    previousSetPos : LREAL; // degrees
    previousSetVelo : LREAL; // degrees/sec
    previousSetAcc : LREAL; // degrees/sec2

    deltaTime : LREAL; // seconds
    
    nextSetPosMax : LREAL;
    nextSetPosMin : LREAL;
    
    nextSetVeloMax : LREAL;
    nextSetVeloMin : LREAL;
    
    nextSetAccMax : LREAL;
    nextSetAccMin : LREAL;
    
    
    lastReceivedDcTime : LINT;
    cycle : INT;
    secondsAfterNewUpdate : LREAL;
    MAX_NUMBER_OF_CYCLES : INT;
    
    minPositionSetpoint : LREAL;
    maxPositionSetpoint : LREAL;
    
END_VAR


// calculate which cycle we are after receiving new updates from the slalib task
IF cycle > MAX_NUMBER_OF_CYCLES THEN 
    cycle := 0; // should not be happening, don't extrapolate
ELSIF  dcTime > lastReceivedDcTime THEN
    // OK we received new values from the slalib task!
    lastReceivedDcTime := dcTime;
    cycle := 0;
ELSE
    cycle := cycle + 1;
END_IF 

secondsAfterNewUpdate := cycle * TIME_TO_LREAL(GLOBAL.config.PLC_FAST_TASK_TIME) / 1000.0;  // TIME_TO_LREAL returns milliseconds!


IF _requestSynchronize THEN    
    physical.PlcToNc.ExtSetPos := physical.NcToPlc.ActPos;
    physical.PlcToNc.ExtSetVelo := 0.0;
    physical.PlcToNc.ExtSetAcc := 0.0;
    
    previousSetPos := physical.PlcToNc.ExtSetPos;
    previousSetVelo := physical.PlcToNc.ExtSetVelo;
    previousSetAcc := physical.PlcToNc.ExtSetAcc;
    
    _requestSynchronize := FALSE;
ELSIF _requestSetPosition THEN
    physical.PlcToNc.ExtSetPos := _requestSetPositionValue;
    physical.PlcToNc.ExtSetVelo := 0.0;
    physical.PlcToNc.ExtSetAcc := 0.0;
    
    previousSetPos := _requestSetPositionValue;
    previousSetVelo := 0.0;
    previousSetAcc := 0.0;
    
    _requestSetPosition := FALSE;      

ELSIF _requestStartTracking THEN
    tracking := TRUE;
    _requestStartTracking := FALSE;
ELSIF _requestStopTracking THEN
    tracking := FALSE;
    _requestStopTracking := FALSE;
ELSE
    
    
    // we expect MAX_VELOCITY and MAX_ACCELERATION to be positive values!
    velocityLimit := ABS(velocityLimit);
    accelerationLimit := ABS(accelerationLimit);
    
    previousSetPos := physical.PlcToNc.ExtSetPos;
    previousSetVelo := physical.PlcToNc.ExtSetVelo;
    previousSetAcc := physical.PlcToNc.ExtSetAcc;
    
    IF tracking THEN
        
        physical.PlcToNc.ExtSetPos  := virtual.NcToPlc.SetPos  + targetPos - trackingStart;
        physical.PlcToNc.ExtSetVelo := virtual.NcToPlc.SetVelo + targetVelo; 
        physical.PlcToNc.ExtSetAcc  := virtual.NcToPlc.SetAcc  + targetAcc;
        
        // The PLC FAST task runs faster than the C++ Slalib task.
        // As a result, the targetPos/targetVelo/targetAcc are updated at a slower rate than the axis setpoints,
        // which means that the axes setpoints versus time look like a "stair" instead of a smooth curve.
        // Therefore, we extrapolate the position setpoint, based on the velocity of the axes
        // The residual position errors are neglegible 
        
        IF cycle > 0 THEN
            // p(t) = p0 + v*t + (a*t^2)/2
            physical.PlcToNc.ExtSetPos := physical.PlcToNc.ExtSetPos 
                                          + targetVelo * secondsAfterNewUpdate
                                          + targetAcc * secondsAfterNewUpdate*secondsAfterNewUpdate / 2.0; 
        END_IF
        
        minPositionSetpoint := minTrackingPositionSetpoint;
        maxPositionSetpoint := maxTrackingPositionSetpoint;
        
    ELSE
        
        physical.PlcToNc.ExtSetPos  := virtual.NcToPlc.SetPos;
        physical.PlcToNc.ExtSetVelo := virtual.NcToPlc.SetVelo; 
        physical.PlcToNc.ExtSetAcc  := virtual.NcToPlc.SetAcc;
        
        minPositionSetpoint := minVirtualPositionSetpoint;
        maxPositionSetpoint := maxVirtualPositionSetpoint;
    END_IF
    
    
    // check if the position limit is reached
    //=======================================================================================
    // we can still go a bit over it, because otherwise the axis would stop very abruptly.
    limitReached := (physical.PlcToNc.ExtSetPos < minPositionSetpoint) OR (physical.PlcToNc.ExtSetPos > maxPositionSetpoint);
    IF limitReached THEN
        physical.PlcToNc.ExtSetPos := LIMIT(minPositionSetpoint, physical.PlcToNc.ExtSetPos, maxPositionSetpoint);
	END_IF
    
    
    
    // Limit the setpoint trajectory!!!!
    //=======================================================================================
    
    deltaTime := TIME_TO_LREAL(GLOBAL.config.PLC_FAST_TASK_TIME) / 1000.0;
    
    // calculate the min/max acceleration for the next setpoint
    nextSetAccMax := accelerationLimit;  // we don't take jerk into account
    nextSetAccMin := -accelerationLimit; // we don't take jerk into account:
    
    // calculate the min/max velocity for the next setpoint
    nextSetVeloMax := LIMIT(-velocityLimit, previousSetVelo + nextSetAccMax * deltaTime, velocityLimit);
    nextSetVeloMin := LIMIT(-velocityLimit, previousSetVelo + nextSetAccMin * deltaTime, velocityLimit);
    
    // calculate the next min/max position
    nextSetPosMax := previousSetPos + nextSetVeloMax * deltaTime;
    nextSetPosMin := previousSetPos + nextSetVeloMin * deltaTime;
    
    // now update the setpoint generator values
    physical.PlcToNc.ExtSetPos  := LIMIT(nextSetPosMin  , physical.PlcToNc.ExtSetPos  , nextSetPosMax);
    physical.PlcToNc.ExtSetVelo := LIMIT(nextSetVeloMin , physical.PlcToNc.ExtSetVelo , nextSetVeloMax);
    physical.PlcToNc.ExtSetAcc  := LIMIT(nextSetAccMin  , physical.PlcToNc.ExtSetAcc  , nextSetAccMax);
    
    // Set the direction
    //===================
    IF physical.PlcToNc.ExtSetPos > physical.NcToPlc.ActPos THEN
        physical.PlcToNc.ExtSetDirection := 1;
    ELSIF physical.PlcToNc.ExtSetPos < physical.NcToPlc.ActPos THEN
        physical.PlcToNc.ExtSetDirection := -1;
    ELSE
        physical.PlcToNc.ExtSetDirection := 0;
    END_IF
    (*
    IF physical.PlcToNc.ExtSetVelo > 0 THEN
        physical.PlcToNc.ExtSetDirection := 1;
    ELSIF physical.PlcToNc.ExtSetVelo < 0 THEN
        physical.PlcToNc.ExtSetDirection := -1;
    ELSE
        physical.PlcToNc.ExtSetDirection := 0;
    END_IF
    *)

END_IF

METHOD stopTracking : BOOL
VAR_INPUT
END_VAR
_requestStopTracking := TRUE;
END_METHOD

METHOD FB_init : BOOL
VAR_INPUT
	bInitRetains : BOOL; // if TRUE, the retain variables are initialized (warm start / cold start)
	bInCopyCode : BOOL;  // if TRUE, the instance afterwards gets moved into the copy code (online change)
END_VAR
IF TIME_TO_LREAL(GLOBAL.config.PLC_FAST_TASK_TIME) > 0 THEN  // watch for division by zero
    MAX_NUMBER_OF_CYCLES := LREAL_TO_INT( TIME_TO_LREAL(GLOBAL.config.SLALIB_TASK_TIME) / TIME_TO_LREAL(GLOBAL.config.PLC_FAST_TASK_TIME) );
END_IF
END_METHOD

METHOD startTracking : BOOL
VAR_INPUT
END_VAR
_requestStartTracking := TRUE;
END_METHOD

METHOD setPosition
VAR_INPUT
    value : LREAL;
END_VAR
_requestSetPosition := TRUE;
_requestSetPositionValue := value;
END_METHOD

METHOD synchronize
VAR_INPUT
END_VAR
_requestSynchronize := TRUE;
END_METHOD

END_FUNCTION_BLOCK

// ---- MTCS/Common/StateMachines/AngularAxis.TcPOU
FUNCTION_BLOCK AngularAxis EXTENDS SM_AngularAxis;
VAR_INPUT
END_VAR
VAR_OUTPUT
END_VAR
VAR
    _testVar : BOOL;
END_VAR

SUPER^();

END_FUNCTION_BLOCK

// ---- MTCS/Axes/Helper/AxesUnlockBrakeHelper.TcPOU
FUNCTION_BLOCK AxesUnlockBrakeHelper
VAR_INPUT
END_VAR
VAR_OUTPUT
END_VAR
VAR_IN_OUT
    unlockBrake : AxesUnlockBrakeProcess;
    driveChannel : AX52XXDriveChannel;
END_VAR
VAR
    _ton : TON;
    _seconds : LREAL;
    _formatString : FB_FormatString;
    _msg : STRING;
END_VAR

IF unlockBrake.isBusy() THEN
    
    IF NOT unlockBrake.isStarted() THEN
        unlockBrake._state := 0;
        unlockBrake.setStarted();
	END_IF
    
    CASE unlockBrake._state OF
        0:
            unlockBrake.setActualStatus('Unlocking brake'); 
            driveChannel.processes.setBrake.start(DriveBrakeStates.BRAKE_FORCE_UNLOCK);
            unlockBrake._state := 1;
        1:
            IF driveChannel.processes.setBrake.isIdle() THEN
                IF driveChannel.processes.setBrake.isGood() THEN
                    _ton(IN := FALSE);
                    _ton(IN := TRUE, PT := LREAL_TO_TIME(unlockBrake.get.seconds * 1000.0));
                    unlockBrake._state := 2;
                ELSE
                    unlockBrake._state := 999;
                    unlockBrake.setActualStatus('Could not change brake to FORCE UNLOCK'); 
				END_IF
			END_IF
        2:
            _ton(IN := TRUE);
            IF _ton.Q THEN
                unlockBrake._state := 3;
            ELSE
                _seconds := TIME_TO_LREAL(_ton.ET) / 1000.0;
                _formatString(sFormat := 'Waiting for %.1fs...', arg1 := F_LREAL(_seconds), sOut => _msg);
                unlockBrake.setActualStatus(_msg); 
			END_IF
        3:
            unlockBrake.setActualStatus('Setting brake to auto'); 
            driveChannel.processes.setBrake.start(DriveBrakeStates.BRAKE_AUTOMATIC);
            unlockBrake._state := 4;
        4:
            IF driveChannel.processes.setBrake.isIdle() THEN
                IF driveChannel.processes.setBrake.isGood() THEN
                    unlockBrake.setActualStatus('Done, brake set to AUTO again'); 
                    unlockBrake._state := 1000;
                ELSE
                    unlockBrake.setActualStatus('Could not change brake to AUTO!!! Brake is still UNLOCKED!!!'); 
                    unlockBrake._state := 999;
				END_IF
			END_IF

        999:
            unlockBrake.setBad();
            unlockBrake.setFinished();
        1000:
            unlockBrake.setGood();
            unlockBrake.setFinished();
        
    END_CASE
    
END_IF

END_FUNCTION_BLOCK

// ---- MTCS/Common/StateMachines/AX52XXDriveChannel.TcPOU
FUNCTION_BLOCK AX52XXDriveChannel EXTENDS SM_AX52XXDriveChannel
VAR_INPUT
END_VAR
VAR_OUTPUT
END_VAR
VAR
    _pointerToAxisRef : POINTER TO AXIS_REF := 0;
    _SoERead : FB_SoERead;
    _SoEWrite : FB_SoEWrite;
    _SoEReset : FB_SoEReset;
	_safetyErrorAckTon: TON;
END_VAR

_update();

isInSafetate := safetyOptionState.0;

_updating();
_reading();
_writing();
_resetting();
_settingBrake();
_acknowledgeSafetyError();

_update();

METHOD _resetting
VAR_INPUT
END_VAR

IF processes.reset.isBusy() THEN
    
    IF NOT processes.reset.isStarted() THEN
        processes.reset._state := 0;
        processes.reset.setStarted();
	END_IF
    
    CASE processes.reset._state OF
        0:  
            processes.reset.setActualStatus('Resetting any errors');
            // Execute must be FALSE first, to make sure we can create a rising edge
            _SoEReset(
                NetId := '',
                Execute := FALSE,
                Axis := _pointerToAxisRef^);
            _SoEReset(
                NetId := '',
                Execute := TRUE,
                Axis := _pointerToAxisRef^,
                Timeout := T#10S); // From Beckhoff help pages: "The timeout time must be 10s, because the reset can take up to 10s."
            processes.reset._state := 1;
        1:
            _SoEReset(
                NetId := '',
                Execute := TRUE,
                Axis := _pointerToAxisRef^,
                Timeout := T#10S);
            
            IF _SoEReset.Error THEN
                processes.reset.setActualStatus(
                        CONCAT(    
                               CONCAT('Reset error: AdsErrId=', UINT_TO_STRING(_SoEReset.AdsErrId)), 
                               CONCAT(' SercosErrId=', UINT_TO_STRING(_SoEReset.SercosErrId))
                        )
                );
                processes.reset.adsErrorId := _SoEReset.AdsErrId;
                processes.reset.sercosErrorId := _SoEReset.SercosErrId;
                processes.reset._state := 999;
            ELSIF NOT _SoEReset.Busy THEN
                // ok done!
                processes.reset._state := 1000;
            END_IF
        999:
            // error!
            processes.reset.setBad();
            processes.reset.setFinished();
        1000:
            // all done!
            processes.reset.setActualStatus('Reset finished');
            processes.reset.setGood();
            processes.reset.setFinished();
    
	END_CASE
        

END_IF
END_METHOD

METHOD _reading
VAR_INPUT
END_VAR
VAR
    valueAddress : PVOID;
END_VAR
IF processes.read.statuses.busyStatus.busy THEN
    
    IF processes.read.get.noOfBytes = 1 THEN
        valueAddress := ADR(processes.read.value1Byte);
        processes.read.setGood();
    ELSIF processes.read.get.noOfBytes = 2 THEN
        valueAddress := ADR(processes.read.value2Bytes);
        processes.read.setGood();
    ELSIF processes.read.get.noOfBytes = 4 THEN
        valueAddress := ADR(processes.read.value4Bytes);
        processes.read.setGood();
    ELSE
        processes.read.setBad();
        processes.read.setFinished();
	END_IF
    
    IF _pointerToAxisRef = 0 THEN
        processes.read.setActualStatus('Internal bug: axis_ref not set');
        processes.read.setBad();
        processes.read.setFinished();
	END_IF
    
    IF processes.read.statuses.healthStatus.good THEN
         
        IF NOT processes.read.statuses.startedStatus.started THEN
            // make sure we get a rising edge
            _SoERead(Execute := FALSE, Axis:= _pointerToAxisRef^);
            
            (* execute the SoE read command *)
            _SoERead(
                NetId    := '',
                Idn      :=  processes.read.get.index,
                Element  := EC_SOE_ELEMENT_VALUE,
                pDstBuf  := valueAddress,
                BufLen   := processes.read.get.noOfBytes,
                Execute  := TRUE,
                Timeout  := DEFAULT_ADS_TIMEOUT,
                Axis     := _pointerToAxisRef^);
            
             processes.read.setStarted();
             
		END_IF
        
       (* Make sure the Execute input is reset *)
        _SoERead(Execute := FALSE, Axis:= _pointerToAxisRef^);
        
        (* update the health status *)
        SUPER^.processes.read.statuses.healthStatus(isGood := NOT _SoERead.Error);
        
        (* update the busy status *)
        SUPER^.processes.read.statuses.busyStatus(isBusy := _SoERead.Busy);
        
        (* update the error ID *)
        SUPER^.processes.read.adsErrorId := _SoERead.AdsErrId;
        SUPER^.processes.read.sercosErrorId := _SoERead.SercosErrId;
             
	END_IF
 
END_IF
END_METHOD

METHOD _acknowledgeSafetyError
VAR_INPUT
END_VAR

VAR
END_VAR

IF processes.acknowledgeSafetyError.isBusy() THEN
    
    IF NOT processes.acknowledgeSafetyError.isStarted() THEN
        processes.acknowledgeSafetyError._state := 0;
        processes.acknowledgeSafetyError.setStarted();
	END_IF
    
    CASE processes.acknowledgeSafetyError._state OF
        0:  
            processes.acknowledgeSafetyError.setActualStatus('Commanding safety card');
            safetyErrorAck := TRUE;
            _safetyErrorAckTon(IN := FALSE);
            
            processes.acknowledgeSafetyError._state := 1;
        1:
            _safetyErrorAckTon(IN := TRUE, PT := T#0.3S);
            IF _safetyErrorAckTon.Q THEN
                processes.acknowledgeSafetyError._state := 2;
            END_IF
        2:
            safetyErrorAck := FALSE;
            _safetyErrorAckTon(IN := FALSE);
            processes.acknowledgeSafetyError._state := 3;
        3:
            _safetyErrorAckTon(IN := TRUE, PT := T#0.3S);
            IF _safetyErrorAckTon.Q THEN
                processes.acknowledgeSafetyError._state := 4;
            END_IF
        4:
            safetyErrorAck := TRUE;
            _safetyErrorAckTon(IN := FALSE);
            processes.acknowledgeSafetyError._state := 5;
        5:
            _safetyErrorAckTon(IN := TRUE, PT := T#0.3S);
            IF _safetyErrorAckTon.Q THEN
                processes.acknowledgeSafetyError._state := 6;
            END_IF
        6:
            safetyErrorAck := FALSE;
            _safetyErrorAckTon(IN := FALSE);
            _safetyErrorAckTon(IN := TRUE, PT := T#1S);
            processes.acknowledgeSafetyError._state := 7;
        7:
            _safetyErrorAckTon(IN := TRUE, PT := T#1S);
            IF _safetyErrorAckTon.Q THEN
                IF isInSafetate THEN
                    processes.acknowledgeSafetyError._state := 999;
                    processes.acknowledgeSafetyError.setActualStatus('Safe state persists!');
                ELSE
                    processes.acknowledgeSafetyError._state := 1000;
                    processes.acknowledgeSafetyError.setActualStatus('Drive unblocked by safety');
                END_IF
            
			END_IF
        999:
            // error!
            processes.acknowledgeSafetyError.setBad();
            processes.acknowledgeSafetyError.setFinished();
        1000:
            // all done!
            processes.acknowledgeSafetyError.setGood();
            processes.acknowledgeSafetyError.setFinished();
    
        END_CASE
            

END_IF
END_METHOD

METHOD _updating
VAR_INPUT
END_VAR

IF processes.update.isBusy() THEN
    
    IF NOT processes.update.isStarted() THEN
        processes.update._state := 0;
        processes.update.setStarted();
	END_IF
    
    CASE processes.update._state OF
        0:  
            processes.update.setActualStatus('Reading P-0-0092 Configured channel peak current');
            processes.read.start(index := P_0_IDN + 92, noOfBytes := 4);
            processes.update._state := 1;
        1:
            IF processes.read.isIdle() THEN
                IF processes.read.isGood() THEN
                    channelPeakCurrent(newAmpsValue := UDINT_TO_LREAL(processes.read.value4Bytes) / 1000.0);
                    processes.update._state := 2;
                ELSE
                    processes.update.setActualStatus('Could not read P-0-0092');
                    processes.update._state := 999;
				END_IF
            END_IF
        2:
            processes.update.setActualStatus('Reading P-0-0093 Configured channel current');
            processes.read.start(index := P_0_IDN + 93, noOfBytes := 4);
            processes.update._state := 3;
        3:
            IF processes.read.isIdle() THEN
                IF processes.read.isGood() THEN
                    channelRatedCurrent(newAmpsValue := UDINT_TO_LREAL(processes.read.value4Bytes) / 1000.0);
                    processes.update._state := 4;
                ELSE
                    processes.update.setActualStatus('Could not read P-0-0093');
                    processes.update._state := 999;
				END_IF
            END_IF
        4:  
            processes.update.setActualStatus('Reading P-0-0070 Motor continuous stall torque');
            processes.read.start(index := P_0_IDN + 70, noOfBytes := 2);
            processes.update._state := 5;
        5:
            IF processes.read.isIdle() THEN
                IF processes.read.isGood() THEN
                        continuousStallTorque(newNewtonmeterValue := UINT_TO_LREAL(processes.read.value2Bytes) / 100.0);
                        processes.update._state := 6;
                ELSE
                    processes.update.setActualStatus('Could not read P-0-070');
                    processes.update._state := 999;
				END_IF
            END_IF 
        6:  
            processes.update.setActualStatus('Reading S-0-0111 Motor continuous stall current');
            processes.read.start(index := S_0_IDN + 111, noOfBytes := 4);
            processes.update._state := 7;
        7:
            IF processes.read.isIdle() THEN
                IF processes.read.isGood() THEN
                        continuousStallCurrent(newAmpsValue := UDINT_TO_LREAL(processes.read.value4Bytes) / 1000.0);
                        processes.update._state := 8;
                ELSE
                    processes.update.setActualStatus('Could not read S-0-0111');
                    processes.update._state := 999;
				END_IF
            END_IF
        8:
            // now we can simply calculate the torque constant:
            // but watch for division by zero!!!
            IF continuousStallCurrent.amps.value > 0 THEN
                torqueConstant := continuousStallTorque.newtonmeter.value / continuousStallCurrent.amps.value;
                processes.update._state := 9;
            ELSE
                torqueConstant := 0.0;
                processes.update.setActualStatus('Torque constant cannot be calculated!');
                processes.update._state := 999;
			END_IF
        9:
            processes.update.setActualStatus('Reading S-0-0082 Positive torque limit value');
            processes.read.start(index := S_0_IDN + 82, noOfBytes := 2);
            processes.update._state := 10;
        10:
            IF processes.read.isIdle() THEN
                IF processes.read.isGood() THEN
                        positiveTorqueLimit(
                            newFractionValue := UINT_TO_LREAL(processes.read.value2Bytes) / 1000.0, 
                            maxNewtonmeter   := channelPeakCurrent.amps.value * torqueConstant);
                        processes.update._state := 11;
                ELSE
                    processes.update.setActualStatus('Could not read S-0-0082');
                    processes.update._state := 999;
				END_IF
            END_IF 
        11:  
            processes.update.setActualStatus('Reading S-0-0083 Negative torque limit value');
            processes.read.start(index := S_0_IDN + 83, noOfBytes := 2);
            processes.update._state := 12;
        12:
            IF processes.read.isIdle() THEN
                IF processes.read.isGood() THEN
                        negativeTorqueLimit(
                            newFractionValue := UINT_TO_LREAL(processes.read.value2Bytes) / 1000.0, 
                            maxNewtonmeter   := channelPeakCurrent.amps.value * torqueConstant);
                        processes.update._state := 13;
                ELSE
                    processes.update.setActualStatus('Could not read S-0-0082');
                    processes.update._state := 999;
				END_IF
            END_IF
        13:  
            processes.update.setActualStatus('Reading S-0-0092 Bipolar torque limit value');
            processes.read.start(index := S_0_IDN + 92, noOfBytes := 2);
            processes.update._state := 14;
        14:
            IF processes.read.isIdle() THEN
                IF processes.read.isGood() THEN
                        bipolarTorqueLimit(
                            newFractionValue := UINT_TO_LREAL(processes.read.value2Bytes) / 1000.0, 
                            maxNewtonmeter   := channelPeakCurrent.amps.value * torqueConstant);
                        processes.update._state := 15;
                ELSE
                    processes.update.setActualStatus('Could not read S-0-0092');
                    processes.update._state := 999;
				END_IF
            END_IF       
        15:  
            processes.update.setActualStatus('Reading P-0-0096 Motor control word');
            processes.read.start(index := P_0_IDN + 96, noOfBytes := 2);
            processes.update._state := 16;
        16:
            IF processes.read.isIdle() THEN
                IF processes.read.isGood() THEN
                    IF processes.read.value2Bytes.0 THEN
                       brakeState := DriveBrakeStates.BRAKE_FORCE_LOCK;
                    ELSIF processes.read.value2Bytes.1 THEN
                       brakeState := DriveBrakeStates.BRAKE_FORCE_UNLOCK;
                    ELSE
                       brakeState := DriveBrakeStates.BRAKE_AUTOMATIC;
                    END_IF
                    brakeStateDescription := DriveBrakeStatesToString(brakeState);
                    processes.update._state := 17;
                ELSE
                    processes.update.setActualStatus('Could not read P-0-0096');
                    processes.update._state := 999;
				END_IF
            END_IF     
        17:  
            processes.update.setActualStatus('Reading S-0-0032 Primary operation mode');
            processes.read.start(index := S_0_IDN + 32, noOfBytes := 2);
            processes.update._state := 18;
        18:
            IF processes.read.isIdle() THEN
                IF processes.read.isGood() THEN
                    IF processes.read.value2Bytes = 0 THEN
                       operatingMode := DriveOperatingModes.OPERATING_MODE_NONE;
                    ELSIF    processes.read.value2Bytes = 1
                          OR processes.read.value2Bytes = 32769 THEN
                       operatingMode := DriveOperatingModes.OPERATING_MODE_TORQUE_CONTROL;
                    ELSIF    processes.read.value2Bytes = 2
                          OR processes.read.value2Bytes = 32770 THEN
                       operatingMode := DriveOperatingModes.OPERATING_MODE_VELOCITY_CONTROL;
                    ELSIF    processes.read.value2Bytes = 3
                          OR processes.read.value2Bytes = 4
                          OR processes.read.value2Bytes = 11
                          OR processes.read.value2Bytes = 12
                          OR processes.read.value2Bytes = 32771
                          OR processes.read.value2Bytes = 32772
                          OR processes.read.value2Bytes = 32779
                          OR processes.read.value2Bytes = 32780 THEN
                       operatingMode := DriveOperatingModes.OPERATING_MODE_POSITION_CONTROL;
                    ELSE
                       operatingMode := DriveOperatingModes.OPERATING_MODE_NONE;
                    END_IF
                    operatingModeDescription := DriveOperatingModesToString(operatingMode);
                    processes.update._state := 19;
                ELSE
                    processes.update.setActualStatus('Could not read S-0-0032');
                    processes.update._state := 999;
				END_IF
            END_IF
        19:
            // all done
            processes.update._state := 1000;
        999:
            // error!
            processes.update.setBad();
            processes.update.setFinished();
        1000:
            // all done!
            processes.update.setActualStatus('Updated');
            processes.update.setGood();
            processes.update.setFinished();
    
    
	END_CASE
        

END_IF
END_METHOD

METHOD _settingBrake
VAR_INPUT
END_VAR
VAR
    ctrlWord : WORD := 0;
END_VAR

IF processes.setBrake.isBusy() THEN
    
    IF NOT processes.setBrake.isStarted() THEN
        processes.setBrake._state := 0;
        processes.setBrake.setStarted();
	END_IF
    
    CASE processes.setBrake._state OF
        0:  
            processes.setBrake.setActualStatus(CONCAT('Setting brake ', DriveBrakeStatesToString(processes.setBrake.get.newState)));          
            CASE processes.setBrake.get.newState OF
               DriveBrakeStates.BRAKE_FORCE_LOCK:
                    ctrlWord.0 := TRUE;
                    ctrlWord.1 := FALSE;
               DriveBrakeStates.BRAKE_FORCE_UNLOCK:
                    ctrlWord.0 := FALSE;
                    ctrlWord.1 := TRUE;
               DriveBrakeStates.BRAKE_AUTOMATIC:
                    ctrlWord.0 := FALSE;
                    ctrlWord.1 := FALSE;
            END_CASE
            
            processes.write.start(index := P_0_IDN + 96, noOfBytes := 2, value1Byte := 0, value2Bytes := ctrlWord, value4Bytes := 0);
            processes.setBrake._state := 1;
        1:
            IF processes.write.isIdle() THEN
                IF processes.write.isGood() THEN
                    processes.setBrake._state := 2;
                ELSE
                    processes.setBrake.setActualStatus('Could not write P-0-0096');
                    processes.setBrake._state := 999;
				END_IF
            END_IF    
        2:  
            processes.setBrake.setActualStatus('Reading P-0-0096 Motor control word');
            processes.read.start(index := P_0_IDN + 96, noOfBytes := 2);
            processes.setBrake._state := 3;
        3:
            IF processes.read.isIdle() THEN
                IF processes.read.isGood() THEN
                    IF processes.read.value2Bytes.0 THEN
                       brakeState := DriveBrakeStates.BRAKE_FORCE_LOCK;
                    ELSIF processes.read.value2Bytes.1 THEN
                       brakeState := DriveBrakeStates.BRAKE_FORCE_UNLOCK;
                    ELSE
                       brakeState := DriveBrakeStates.BRAKE_AUTOMATIC;
                    END_IF
                    brakeStateDescription := DriveBrakeStatesToString(brakeState);
                    processes.setBrake._state := 1000;
                ELSE
                    processes.setBrake.setActualStatus('Could not read P-0-0096');
                    processes.setBrake._state := 999;
				END_IF
            END_IF     
            

        999:
            // error!
            processes.setBrake.setBad();
            processes.setBrake.setFinished();
        1000:
            // all done!
            processes.setBrake.setActualStatus(CONCAT('Brake now ', brakeStateDescription));
            processes.setBrake.setGood();
            processes.setBrake.setFinished();
    
	END_CASE
        

END_IF
END_METHOD

METHOD _update
VAR_INPUT
END_VAR
SUPER^();

IF statuses.healthStatus.good THEN
    IF statuses.busyStatus.idle THEN
        IF isInSafetate THEN
            actualStatus := 'In safe state';
        ELSE
            actualStatus := 'Idle';
        END_IF
    ELSIF statuses.busyStatus.busy THEN
        actualStatus := 'Busy';
    ELSE
        actualStatus := 'Good';
    END_IF
ELSIF statuses.healthStatus.warning THEN
    IF isInSafetate THEN
        actualStatus := 'SAFE STATE';
    ELSE
        actualStatus := 'Warning';
	END_IF
ELSIF statuses.healthStatus.bad THEN
    IF errorC1D <> 0 THEN
        actualStatus := CONCAT(CONCAT('C1D error (id: ', INT_TO_STRING(errorC1D)), ')');
    ELSIF isInSafetate THEN
        actualStatus := 'SAFE STATE';
    ELSE
        actualStatus := 'ERROR';
	END_IF
ELSE
    actualStatus := '';
END_IF
END_METHOD

METHOD setInternalAxisRef
VAR_INPUT
    pointerToAxisRef : POINTER TO AXIS_REF;
END_VAR
_pointerToAxisRef := pointerToAxisRef;
END_METHOD

METHOD _writing
VAR_INPUT
END_VAR
VAR
    srcAddress : PVOID;
END_VAR
IF processes.write.statuses.busyStatus.busy THEN
    
    IF processes.write.get.noOfBytes = 1 THEN
        srcAddress := ADR(processes.write.get.value1Byte);
        processes.write.setGood();
    ELSIF processes.write.get.noOfBytes = 2 THEN
        srcAddress := ADR(processes.write.get.value2Bytes);
        processes.write.setGood();
    ELSIF processes.write.get.noOfBytes = 4 THEN
        srcAddress := ADR(processes.write.get.value4Bytes);
        processes.write.setGood();
    ELSE
        processes.write.setBad();
        processes.write.setFinished();
	END_IF
     
    IF _pointerToAxisRef = 0 THEN
        processes.write.setActualStatus('Internal bug: axis_ref not set');
        processes.write.setBad();
        processes.write.setFinished();
	END_IF
    
    IF processes.write.statuses.healthStatus.good THEN
         
        IF NOT processes.write.statuses.startedStatus.started THEN
        
            // make sure we get a rising edge
            _SoEWrite(Execute := FALSE, Axis:= _pointerToAxisRef^);
            (* execute the SoE write command *)
            _SoEWrite(
                NetId    := '',
                Idn      :=  processes.write.get.index,
                Element  := EC_SOE_ELEMENT_VALUE,
                pSrcBuf  := srcAddress,
                BufLen   := processes.write.get.noOfBytes,
                Execute  := TRUE,
                Timeout  := DEFAULT_ADS_TIMEOUT,
                Axis     := _pointerToAxisRef^);
            
             processes.write.setStarted();
        ELSE
            // make sure the Exectute input is reset
            _SoEWrite(Execute := FALSE, Axis:= _pointerToAxisRef^);
        
        (* update the health status *)
        SUPER^.processes.write.statuses.healthStatus(isGood := NOT _SoEWrite.Error);
        
        (* update the busy status *)
        SUPER^.processes.write.statuses.busyStatus(isBusy := _SoEWrite.Busy);
        
        (* update the error ID *)
        SUPER^.processes.write.adsErrorId := _SoEWrite.AdsErrId;
        SUPER^.processes.write.sercosErrorId := _SoEWrite.SercosErrId;
		END_IF
        
             
	END_IF
    

 
END_IF
END_METHOD

END_FUNCTION_BLOCK

// ---- MTCS/Common/StateMachines/Current.TcPOU
FUNCTION_BLOCK Current EXTENDS SM_Current
VAR_INPUT
END_VAR
VAR_OUTPUT
END_VAR
VAR
    _testVar : INT;
END_VAR

SUPER^();

END_FUNCTION_BLOCK

// ---- MTCS/Common/HelperCode/DriveBrakeStatesToString.TcPOU
FUNCTION DriveBrakeStatesToString : STRING
VAR_INPUT
    state : DriveBrakeStates;
END_VAR
VAR
END_VAR

CASE state OF
    
    DriveBrakeStates.BRAKE_AUTOMATIC:
        DriveBrakeStatesToString := 'Automatic';
    DriveBrakeStates.BRAKE_FORCE_LOCK:
        DriveBrakeStatesToString := 'Forced LOCK';
    DriveBrakeStates.BRAKE_FORCE_UNLOCK:
        DriveBrakeStatesToString := 'Forced UNLOCK';

END_CASE

END_FUNCTION

// ---- MTCS/Common/HelperCode/DriveOperatingModesToString.TcPOU
FUNCTION DriveOperatingModesToString : STRING
VAR_INPUT
    mode : DriveOperatingModes;
END_VAR
VAR
END_VAR

CASE mode OF
    
    DriveOperatingModes.OPERATING_MODE_NONE:
        DriveOperatingModesToString := 'None';
    DriveOperatingModes.OPERATING_MODE_TORQUE_CONTROL:
        DriveOperatingModesToString := 'Torque control';
    DriveOperatingModes.OPERATING_MODE_VELOCITY_CONTROL:
        DriveOperatingModesToString := 'Velocity control';
    DriveOperatingModes.OPERATING_MODE_POSITION_CONTROL:
        DriveOperatingModesToString := 'Position control';

END_CASE

END_FUNCTION

// ---- MTCS/Common/StateMachines/Force.TcPOU
FUNCTION_BLOCK Force EXTENDS SM_Force
VAR_INPUT
END_VAR
VAR_OUTPUT
END_VAR
VAR
    _testVar : INT;
END_VAR

SUPER^();

END_FUNCTION_BLOCK

// ---- MTCS/Axes/Helper/HMS_TO_DEG.TcPOU
FUNCTION HMS_TO_DEG : LREAL
VAR_INPUT
    positive : BOOL;
    hours : LREAL;
    minutes : LREAL;
    seconds : LREAL;
END_VAR
VAR
END_VAR

HMS_TO_DEG := (hours/24.0 + minutes/(24.0*60.0) + seconds/(24.0*60.0*60.0)) * 360.0;

IF NOT positive THEN
    HMS_TO_DEG := -HMS_TO_DEG;
END_IF

END_FUNCTION

// ---- MTCS/Axes/Helper/DMS_TO_DEG.TcPOU
FUNCTION DMS_TO_DEG : LREAL
VAR_INPUT
    positive : BOOL;
    degrees : LREAL;
    minutes : LREAL;
    seconds : LREAL;
END_VAR
VAR
END_VAR

DMS_TO_DEG := degrees + minutes/60.0 + seconds/3600.0;

IF NOT positive THEN
    DMS_TO_DEG := -DMS_TO_DEG;
END_IF

END_FUNCTION

// ---- MTCS/Axes/Helper/AverageAndRmsCalculator.TcPOU
FUNCTION_BLOCK AverageAndRmsCalculator
VAR_INPUT
    in : LREAL;
END_VAR
VAR_OUTPUT
    avg : LREAL;
    rms : LREAL;
END_VAR
VAR
	_executeMovingAverage : BOOL;
    _ctrl_moving_avg : FB_CTRL_MOVING_AVERAGE;
    _PARAMS : ST_CTRL_MOVING_AVERAGE_PARAMS;
    _array : ARRAY [1..100] OF LREAL;
    
    i : INT := 0;
    sumOfSquares : LREAL := 0.0;
END_VAR


_params.nSamplesToFilter  := 100;
_params.tCtrlCycleTime    := GLOBAL.config.PLC_CTRL_TIME;
_params.tTaskCycleTime    := GLOBAL.config.PLC_TASK_TIME;
_params.pWorkArray_ADR    := ADR(_array);
_params.nWorkArray_SIZEOF := SIZEOF(_array);

IF _executeMovingAverage <> GLOBAL.config.PLC_TASK_FLIP THEN
	_executeMovingAverage := GLOBAL.config.PLC_TASK_FLIP;
	_ctrl_moving_avg(
		fIn             := in,
		fManSyncValue   := 0.0,
		bSync           := FALSE,
		eMode           := E_CTRL_MODE.eCTRL_MODE_ACTIVE,
		bHold           := FALSE,
		stParams        := _params);
    
    sumOfSquares := 0.0;
    FOR i := 1 TO 100 BY 1 DO
        sumOfSquares := sumOfSquares + _array[i]*_array[i];
    END_FOR 
    
    avg := _ctrl_moving_avg.fOut;
    rms := SQRT(sumOfSquares / 100.0);
END_IF

END_FUNCTION_BLOCK

// ---- MTCS/Axes/Helper/AxesCalculateLidaAveragePosition.TcPOU
FUNCTION AxesCalculateLidaAveragePosition : LREAL
VAR_INPUT
    lida1Position : LREAL;
    lida2Position : LREAL;
    lida3Position : LREAL;
    lida4Position : LREAL;
    useLida1 : BOOL;
    useLida2 : BOOL;
    useLida3 : BOOL;
    useLida4 : BOOL;
END_VAR
VAR_OUTPUT
    error : BOOL;
END_VAR
VAR
    sumOfPositions : LREAL := 0.0;
    noOfLidasUsed : INT := 0;
END_VAR

IF useLida1 THEN
    noOfLidasUsed := noOfLidasUsed + 1;
    sumOfPositions := sumOfPositions + lida1Position;
END_IF

IF useLida2 THEN
    noOfLidasUsed := noOfLidasUsed + 1;
    sumOfPositions := sumOfPositions + lida2Position;
END_IF

IF useLida3 THEN
    noOfLidasUsed := noOfLidasUsed + 1;
    sumOfPositions := sumOfPositions + lida3Position;
END_IF

IF useLida4 THEN
    noOfLidasUsed := noOfLidasUsed + 1;
    sumOfPositions := sumOfPositions + lida4Position;
END_IF

// watch for division by zero!
error := noOfLidasUsed = 0;

IF error THEN
    AxesCalculateLidaAveragePosition := 0.0;
ELSE
    AxesCalculateLidaAveragePosition := sumOfPositions / noOfLidasUsed;
END_IF

END_FUNCTION

// ---- MTCS/Axes/Helper/AxesLidaValueToPosition.TcPOU
FUNCTION AxesLidaValueToPosition : LREAL
VAR_INPUT
    id : AxesIds;
    encoderValue : UDINT; 
    invert : BOOL;
END_VAR
VAR
    BITS_PER_TELESCOPE_REVOLUTION : LREAL;
    ENCODER_DIRECTION_INVERSE : BOOL;
END_VAR



IF GLOBAL.config.SIMULATION_ACTIVE THEN
    
    CASE id OF
        AxesIds.AZI:
            BITS_PER_TELESCOPE_REVOLUTION := 3000    // bits per simulation encoder revolution
                                             * 4     // quadrature interpolation
                                             * 1440; // reduction
        AxesIds.ELE:
            BITS_PER_TELESCOPE_REVOLUTION := 3000    // bits per simulation encoder revolution
                                             * 4     // quadrature interpolation
                                             * 1440; // reduction
	END_CASE
ELSE
    
    CASE id OF
        AxesIds.AZI:
            BITS_PER_TELESCOPE_REVOLUTION := 45000    // marks (lines, ticks) on the linear Heidenhain encoder
                                             * 100    // Heidenhain EXE interpolation
                                             * 4;     // quadrature interpolation
        AxesIds.ELE:
            BITS_PER_TELESCOPE_REVOLUTION := 45000    // marks (lines, ticks) on the linear Heidenhain encoder
                                             * 100    // Heidenhain EXE interpolation
                                             * 4;     // quadrature interpolation
	END_CASE

END_IF

    
// we go from unsigned raw value, to signed position in degrees:
IF encoderValue.31 THEN
    AxesLidaValueToPosition := (UDINT_TO_LREAL(encoderValue) - 4294967296) / BITS_PER_TELESCOPE_REVOLUTION * 360.0;  // (rawValue bits - 2**32 bits) / BITS_PER_TELESCOPE_REVOLUTION * 360.0 degrees
ELSE
    AxesLidaValueToPosition := UDINT_TO_LREAL(encoderValue) / BITS_PER_TELESCOPE_REVOLUTION * 360.0; // rawValue bits / BITS_PER_TELESCOPE_REVOLUTION * 360.0 degrees
END_IF

IF invert THEN
    AxesLidaValueToPosition := -AxesLidaValueToPosition;
END_IF

END_FUNCTION

// ---- MTCS/Axes/Helper/AxesSSIValueToPosition.TcPOU
FUNCTION AxesSSIValueToPosition : LREAL
VAR_INPUT
    reduction : LREAL;
    encoderValue : UDINT;
    zeroOffset : LREAL;
END_VAR
VAR
    BITS_PER_ENCODER_REVOLUTION : LREAL := 8192; // 13-bit
    ENCODER_BIT_RANGE : LREAL := 33554432; // 25-bit
END_VAR

// we go from unsigned raw value, to signed position in degrees:
IF encoderValue.24 THEN
    AxesSSIValueToPosition := (UDINT_TO_LREAL(encoderValue) - ENCODER_BIT_RANGE) / BITS_PER_ENCODER_REVOLUTION / reduction * 360.0 + zeroOffset;
ELSE
    AxesSSIValueToPosition := UDINT_TO_LREAL(encoderValue) / BITS_PER_ENCODER_REVOLUTION / reduction * 360.0 + zeroOffset;
END_IF

END_FUNCTION

// ---- MTCS/Axes/Helper/AxesMoveOutOfLimitSwitchHelper.TcPOU
FUNCTION_BLOCK AxesMoveOutOfLimitSwitchHelper
VAR_INPUT
    positiveLimitSwitchError : BOOL;
    negativeLimitSwitchError : BOOL;
    positiveLimitSwitchInput : SINT;
    negativeLimitSwitchInput : SINT;
    moveOutOfLimitSwitchDistance : LREAL;
END_VAR
VAR_OUTPUT
END_VAR
VAR_IN_OUT
    setpointGenerator : AxesExternalSetpointGenerator;
    moveOutOfLimitSwitch : AxesMoveOutOfLimitSwitchProcess;
    moveRelative : AxesMoveRelativeProcess;
    powerOn : AxesPowerOnProcess;
    reset : Process;
    virtual : AngularAxis;
    physical : AngularAxis;
    driveChannel : AX52XXDriveChannel;
END_VAR
VAR
    offset : SINT;
    forceValue : DWORD;
    relativeMoveDistance : LREAL;
END_VAR


// see documentation on P-0-0805 Force digital inputs!!!


IF moveOutOfLimitSwitch.isBusy() THEN
    
    CASE moveOutOfLimitSwitch.get.switch OF
        LimitSwitches.POSITIVE_LIMIT_SWITCH:
            offset := positiveLimitSwitchInput * 2;
            relativeMoveDistance := -ABS(moveOutOfLimitSwitchDistance);
        LimitSwitches.NEGATIVE_LIMIT_SWITCH:
            offset := negativeLimitSwitchInput * 2;
            relativeMoveDistance := ABS(moveOutOfLimitSwitchDistance);
    END_CASE

    IF NOT moveOutOfLimitSwitch.isStarted() THEN
        moveOutOfLimitSwitch._state := 0;
        moveOutOfLimitSwitch.setStarted();
	END_IF
    
    CASE moveOutOfLimitSwitch._state OF
        0:
            moveOutOfLimitSwitch.setActualStatus('Moving out of limit switch');
            
            forceValue := CSETBIT32( inVal32 := forceValue, bitNo := offset     , bitVal := TRUE);
            forceValue := CSETBIT32( inVal32 := forceValue, bitNo := offset + 1 , bitVal := FALSE);
            
            driveChannel.processes.write.start(
                    index       := P_0_IDN + 805, 
                    noOfBytes   := 4, 
                    value1Byte  := 0, 
                    value2Bytes := 0, 
                    value4Bytes := DWORD_TO_UDINT(forceValue));
                    
            moveOutOfLimitSwitch._state := 1;
        1:
            IF  driveChannel.processes.write.isIdle() THEN
                IF driveChannel.processes.write.isGood() THEN
                    moveOutOfLimitSwitch._state := 2;
                ELSE
                    moveOutOfLimitSwitch.setActualStatus('Could not force the limit switch input');
                    moveOutOfLimitSwitch._state := 999;
				END_IF
			END_IF
        2:
            // now we can reset the error
            reset.start();
            moveOutOfLimitSwitch._state := 3;
        3:
            IF reset.isIdle() THEN
                IF reset.isGood() THEN
                    moveOutOfLimitSwitch._state := 4;
                ELSE
                    moveOutOfLimitSwitch.setActualStatus('Could not reset the axis');
                    moveOutOfLimitSwitch._state := 999;
				END_IF
			END_IF
        4:
            // make sure the axis is powered on
            powerOn.start();
            moveOutOfLimitSwitch._state := 5;
        5:
            IF powerOn.isIdle() THEN
                IF powerOn.isIdle() THEN
                    moveOutOfLimitSwitch._state := 6;
                ELSE
                    moveOutOfLimitSwitch.setActualStatus('Could not power on the axis');
                    moveOutOfLimitSwitch._state := 999;
				END_IF
			END_IF
        6:
            // try to move out of the limit switch!
            moveRelative.start(
                        units   := AxesMoveUnits.DEGREES, 
                        value   := relativeMoveDistance);
            moveOutOfLimitSwitch._state := 7;
        7:
            IF moveRelative.isIdle() THEN
                IF moveRelative.isGood() THEN
                    moveOutOfLimitSwitch._state := 8;
                ELSE
                    moveOutOfLimitSwitch.setActualStatus('Could not move out');
                    moveOutOfLimitSwitch._state := 999;
                END_IF
            END_IF
        8:
            // now unforce the digital input
            forceValue := CSETBIT32( inVal32 := forceValue, bitNo := offset     , bitVal := FALSE);
            forceValue := CSETBIT32( inVal32 := forceValue, bitNo := offset + 1 , bitVal := FALSE);
            
            
            driveChannel.processes.write.start(
                    index       := P_0_IDN + 805, 
                    noOfBytes   := 4, 
                    value1Byte  := 0, 
                    value2Bytes := 0, 
                    value4Bytes := DWORD_TO_UDINT(forceValue));
            
            moveOutOfLimitSwitch._state := 9;
        9:
            IF  driveChannel.processes.write.isIdle() THEN
                IF driveChannel.processes.write.isGood() THEN
                    moveOutOfLimitSwitch._state := 10;
                ELSE
                    moveOutOfLimitSwitch.setActualStatus('Could not unforce the limit switch input');
                    moveOutOfLimitSwitch._state := 999;
				END_IF
			END_IF
        10:
            IF moveOutOfLimitSwitch.get.switch = LimitSwitches.POSITIVE_LIMIT_SWITCH AND positiveLimitSwitchError THEN
                moveOutOfLimitSwitch.setActualStatus('Positive limit switch still active!');
                moveOutOfLimitSwitch._state := 999;
            ELSIF moveOutOfLimitSwitch.get.switch = LimitSwitches.NEGATIVE_LIMIT_SWITCH AND negativeLimitSwitchError THEN
                moveOutOfLimitSwitch.setActualStatus('Negative limit switch still active!');
                moveOutOfLimitSwitch._state := 999;
            ELSE
                // all done!
                moveOutOfLimitSwitch._state := 1000;
			END_IF
            
        999:
            // error!
            // try to un-force the inputs!!!
            moveOutOfLimitSwitch._state := 9991;
            
        1000:
            moveOutOfLimitSwitch.setActualStatus('Moved out of limit switch');
            // ok done
            moveOutOfLimitSwitch.setFinished();
            moveOutOfLimitSwitch.setGood();
            
            
        9991:
            // unforce the digital input
            forceValue := CSETBIT32( inVal32 := forceValue, bitNo := offset     , bitVal := FALSE);
            forceValue := CSETBIT32( inVal32 := forceValue, bitNo := offset + 1 , bitVal := FALSE);
            
            driveChannel.processes.write.start(
                    index       := P_0_IDN + 805, 
                    noOfBytes   := 4, 
                    value1Byte  := 0, 
                    value2Bytes := 0, 
                    value4Bytes := DWORD_TO_UDINT(forceValue));
            moveOutOfLimitSwitch._state := 9992;
        9992:
            IF driveChannel.processes.write.isIdle() THEN
                moveOutOfLimitSwitch._state := 9993;
			END_IF
        9993:
            // nothing can be done anymore
            moveOutOfLimitSwitch.setBad();
            moveOutOfLimitSwitch.setFinished();
    END_CASE
    
END_IF

END_FUNCTION_BLOCK

// ---- MTCS/Axes/Helper/AxesPowerOffHelper.TcPOU
FUNCTION_BLOCK AxesPowerOffHelper
VAR_INPUT
    pAblAxis : POINTER TO AngularAxis := 0; (* NULL if no anti-backlash axis is available !!!*)
    pAblDriveChannel : POINTER TO AX52XXDriveChannel := 0; (* NULL if no anti-backlash axis is available !!!*)
    pAblSetpointGenerator : POINTER TO AxesTorqueSetpointGenerator := 0; (* NULL if no anti-backlash axis is available !!!*)
END_VAR
VAR_OUTPUT
END_VAR
VAR_IN_OUT
    setpointGenerator : AxesExternalSetpointGenerator;
    powerOff : AxesPowerOffProcess;
    stop     : AxesStopProcess;
    virtual : AngularAxis;
    physical : AngularAxis;
END_VAR
VAR
    timeoutTon : TON;
END_VAR

IF powerOff.isBusy() THEN
    
    IF NOT powerOff.isStarted() THEN
        powerOff.state := 0;
        powerOff.setStarted();
	END_IF
    
    CASE powerOff.state OF
        0:
            // first make sure the axes are stopped
            powerOff.setActualStatus('Stopping the axes');
            stop.start();         
            powerOff.state := 1;
        1:
            IF stop.isIdle() THEN
                IF stop.isGood() THEN
                    // ok, all axes are stopped
                    powerOff.state := 2;
                ELSE
                    powerOff.setActualStatus('Could not stop the axes!');
                    powerOff.state := 999;
                END_IF
            END_IF
        2:
            IF hasAblAxis() THEN
                powerOff.setActualStatus('Removing anti-backlash torque');
                pAblSetpointGenerator^.stop();
                // start a timer
                timeoutTon(IN := FALSE);
                timeoutTon(IN := TRUE, PT := T#3S);
                powerOff.state := 3;
            ELSE
                // skip the next step
                powerOff.state := 4;
			END_IF
        3:
            // wait for the anti-backlash torque to be ramped down
            IF pAblDriveChannel^.torqueCommandValue = 0 THEN
                powerOff.state := 4;
            ELSIF timeoutTon.Q THEN
                powerOff.setActualStatus('Timeout while removing anti-backlash torque');
                powerOff.state := 999;
			END_IF
        4:
            powerOff.setActualStatus('Disabling external setpoint generator');
            IF physical.statuses.extSetGenStatus.enabled THEN
                physical.processes.disableExtSetGen.start();
                // wait at most 1 second for the external setpoint generators to become disabled
                timeoutTon(IN := FALSE);
                timeoutTon(IN := TRUE, PT := T#1S);
                powerOff.state := 5;
            ELSE
                // skip the next step
                powerOff.state := 6;
            END_IF
            
        5:
            timeoutTon(IN := TRUE);
            IF physical.statuses.extSetGenStatus.disabled THEN
                powerOff.state :=6;
            ELSIF timeoutTon.Q THEN
                powerOff.state := 999;
                powerOff.setActualStatus('Could not disable AZI external setpoint generator');
            END_IF
        6:
            IF hasAblAxis() THEN
                powerOff.setActualStatus('Powering off the anti-backlash axis');
                pAblAxis^.processes.power.start(enable := FALSE);
                powerOff.state := 7;
            ELSE
                // skip the next step
                powerOff.state := 8;
			END_IF
        7:
            IF pAblAxis^.processes.power.isIdle() THEN
                IF pAblAxis^.processes.power.isGood() THEN
                    powerOff.state := 8;
                ELSE
                    powerOff.setActualStatus('Could not power off the anti-backlash axis!');
                    powerOff.state := 999;
                END_IF
            END_IF
        8:
            // now power off the other axes
            powerOff.setActualStatus('Powering off the axes');
            virtual.processes.power.start(enable := FALSE);
            physical.processes.power.start(enable := FALSE);
            powerOff.state := 9;
        9:
            IF      virtual.processes.power.isIdle() 
                AND physical.processes.power.isIdle() THEN
                
                IF      virtual.processes.power.isGood() 
                   AND  physical.processes.power.isGood() THEN
                    // ok, all axes are powered off
                    powerOff.state := 1000;
                ELSE
                    powerOff.setActualStatus('Could not power off the axes!');
                    powerOff.state := 999;
                END_IF
            END_IF
        999:
            // error!
            powerOff.setBad();
            powerOff.setFinished();
            // stop all axes
            stop.start();
        1000:
            powerOff.setActualStatus('Powered off');
            // ok done
            powerOff.setFinished();
            powerOff.setGood();
		
    END_CASE
    
END_IF

METHOD hasAblAxis : BOOL
VAR_INPUT
END_VAR
hasAblAxis := (pAblAxis <> 0) AND (pAblDriveChannel <> 0) AND (pAblSetpointGenerator <> 0);
END_METHOD

END_FUNCTION_BLOCK

// ---- MTCS/Axes/Helper/AxesTorqueSetpointGenerator.TcPOU
FUNCTION_BLOCK AxesTorqueSetpointGenerator
VAR_INPUT
    ablMaxTorqueRiseSpeed : LREAL; // Nm/s
    ablMaxTorqueFallSpeed : LREAL; // Nm/s
    maxAccelerationSetpoint : LREAL; // degrees/sec^2
    ablMaxTorque : LREAL; // Nm
    ablMinTorque : LREAL; // Nm
    ablZeroAccTorque : LREAL; // Nm
    ablTorqueOutputOverride : LREAL; // fraction (not percent!)
    aziAndAblSameDirection : BOOL;
    ablPositiveTorque : BOOL;
END_VAR
VAR_OUTPUT
    output : LREAL;
END_VAR
VAR_IN_OUT
    physicalAxis : AngularAxis;
    virtualAxis : AngularAxis;
    ablAxis : AngularAxis;
END_VAR
VAR
    previousTorqueSetpoint : LREAL;
    
    torqueSetpointUnlimited : LREAL;
    torqueSetpointLimitedByMinMaxTorque : LREAL;
    torqueSetpoint : LREAL;
    
    running : BOOL;
    deltaTime : LREAL; // seconds
    torqueChangeUnlimited : LREAL;
    ZERO_TORQUE : LREAL := 0.0;
    
    aziAccelerationSign : INT;
    torqueSign : INT;
END_VAR


deltaTime := TIME_TO_LREAL(GLOBAL.config.PLC_FAST_TASK_TIME) / 1000.0;

IF aziAndAblSameDirection THEN
    aziAccelerationSign := 1;
ELSE
    aziAccelerationSign := -1;
END_IF

IF ablPositiveTorque THEN
    torqueSign := 1;
ELSE
    torqueSign := -1;
END_IF

IF     (physicalAxis.axis_ref.NcToPlc.StateDWord.0 = TRUE) (* first bit = Operational *) 
   AND (ablAxis.axis_ref.NcToPlc.StateDWord.0 = TRUE) (* first bit = Operational *)
   AND running THEN
    
    // axis is operational!
    
    ablMaxTorqueRiseSpeed := ABS(ablMaxTorqueRiseSpeed);
    ablMaxTorqueFallSpeed := ABS(ablMaxTorqueFallSpeed);
    maxAccelerationSetpoint := ABS(maxAccelerationSetpoint);
    
    IF maxAccelerationSetpoint <> 0  THEN
        
        IF physicalAxis.axis_ref.NcToPlc.SetAcc > 0 THEN
            // accelerating
            torqueSetpointUnlimited := ablZeroAccTorque + aziAccelerationSign * ABS(  (ablMaxTorque - ablZeroAccTorque) * (physicalAxis.axis_ref.NcToPlc.SetAcc / maxAccelerationSetpoint)  );
        ELSE
            // decelerating
            torqueSetpointUnlimited := ablZeroAccTorque - aziAccelerationSign * ABS(  (ablMinTorque - ablZeroAccTorque) * (physicalAxis.axis_ref.NcToPlc.SetAcc / maxAccelerationSetpoint)  );
        END_IF
    
    END_IF
    
    
    // limit by the min/max torque values
    // ----------------------------------
    IF torqueSetpointUnlimited > ablMaxTorque THEN
        torqueSetpointLimitedByMinMaxTorque := ablMaxTorque;
    ELSIF torqueSetpointUnlimited < ablMinTorque THEN
        torqueSetpointLimitedByMinMaxTorque := ablMinTorque;
    ELSE
        torqueSetpointLimitedByMinMaxTorque := torqueSetpointUnlimited;
    END_IF

ELSE
    
    torqueSetpointUnlimited := ZERO_TORQUE;
    torqueSetpointLimitedByMinMaxTorque := ZERO_TORQUE;

END_IF

// limit by the rate of torque change
// ----------------------------------


IF deltaTime <> 0 THEN
    torqueChangeUnlimited := (torqueSetpointLimitedByMinMaxTorque - previousTorqueSetpoint) / deltaTime; // Nm/s on the telescope axis
ELSE
    torqueChangeUnlimited := 0.0; // ignore
END_IF

IF torqueChangeUnlimited > ablMaxTorqueRiseSpeed THEN
    torqueSetpoint := previousTorqueSetpoint + ablMaxTorqueRiseSpeed * deltaTime;
ELSIF torqueChangeUnlimited < - ablMaxTorqueFallSpeed THEN
    torqueSetpoint := previousTorqueSetpoint - ablMaxTorqueFallSpeed * deltaTime;
ELSE
    torqueSetpoint := torqueSetpointLimitedByMinMaxTorque;
END_IF

// send the new setpoint to the drive
// ----------------------------------
output := torqueSetpoint * ablTorqueOutputOverride * torqueSign;


// finally, update the previousTorqueSetpoint for the next cycle
// -------------------------------------------------------------
previousTorqueSetpoint := torqueSetpoint;

METHOD start
VAR_INPUT
END_VAR
running := TRUE;
END_METHOD

METHOD stop
VAR_INPUT
END_VAR
running := FALSE;
END_METHOD

END_FUNCTION_BLOCK

// ---- MTCS/Axes/Helper/AxesHomingHelper.TcPOU
FUNCTION_BLOCK AxesHomingHelper
VAR_INPUT
    id : AxesIds;
    homingStartAbsEncPosition : LREAL;
    homingVelocity : LREAL;
    homingRange : LREAL;
    homingGotoStartVelocity : LREAL;
    homingHomePosition : LREAL;
    absoluteEncoderPosition : LREAL;
    lidasInvert : BOOL;
    lidaAveragePosition : LREAL;
    lida1Position : LREAL;
    pLida1 : POINTER TO IncrementalEncoder := 0;
    pLida2 : POINTER TO IncrementalEncoder := 0;
    pLida3 : POINTER TO IncrementalEncoder := 0;
    pLida4 : POINTER TO IncrementalEncoder := 0;
END_VAR
VAR_OUTPUT
END_VAR
VAR_IN_OUT
    setpointGenerator : AxesExternalSetpointGenerator;
    doHoming : AxesDoHomingProcess;
    stop     : AxesStopProcess;
    setPosition  : AxesSetpositionProcess;
    virtual : AngularAxis;
    physical : AngularAxis;
END_VAR
VAR
    homeTon : TON;
    
    lida1PositionAfterZeroing : LREAL;
    truePositionAfterZeroing : LREAL;
    trueValueAfterZeroing : UDINT;
END_VAR

IF doHoming.isBusy() THEN
    
    IF NOT doHoming.isStarted() THEN
        doHoming.state := 0;
        doHoming.setStarted();
	END_IF
    
    CASE doHoming.state OF
        0:
            doHoming.setActualStatus('Now homing');
            stop.start();
            doHoming.state := 1;
        1:
            IF stop.isIdle() THEN
                IF stop.isGood() THEN
                    // ok, the axes are stopped
                    doHoming.state := 2;
                ELSE
                    doHoming.setActualStatus('Could not stop the axes');
                    doHoming.state := 999;
				END_IF
			END_IF
        2:
            // verify the axis
            IF NOT physical.axis_ref.Status.ExtSetPointGenEnabled THEN
                doHoming.setActualStatus('External setpoint generator disabled! Power on needed!');
                doHoming.state := 999;
            ELSIF physical.axis_ref.Status.Disabled OR virtual.axis_ref.Status.Disabled THEN
                doHoming.setActualStatus('Axis is disabled! Power on needed!');
                doHoming.state := 999;
            ELSIF NOT hasLida1() THEN
                doHoming.setActualStatus('At least one LIDA is needed!');
            ELSE
                doHoming.state := 3;
			END_IF
        3:
            // reset the homing flag
            physical.processes.resetCalibration.start();
            // stop monitoring slip between the external encoder and the motor encoder
            doHoming.state := 4;
        4:
            IF physical.processes.resetCalibration.isIdle() THEN
                IF physical.processes.resetCalibration.isGood() THEN
                    doHoming.state := 5;
                ELSE
                    doHoming.setActualStatus('Could not reset the calibration flag');
                    doHoming.state := 999;
				END_IF
			END_IF
        5:
            // disable the 'enableLatchC' output, so we can turn in on further on
            // When enableLatchC will be set to TRUE (further on), then the latchCValid flag will be raised when the C signal gets activated, in other words, when the counter gets reset
            pLida1^.updateEnableLatchC(FALSE);
            doHoming.setActualStatus('Moving to the homing start');
            virtual.processes.moveRelative.start(
                distance := homingStartAbsEncPosition - absoluteEncoderPosition,
                maxVelocity := homingGotoStartVelocity);
            doHoming.state := 6;
        6:
             // wait for the positioning to be finished
             IF virtual.processes.moveRelative.isIdle() THEN
                 IF virtual.processes.moveRelative.isGood() THEN
                    doHoming.state := 7;
                 ELSE
                    doHoming.setActualStatus('Could not move to homing start');
                    doHoming.state := 999;
				 END_IF
			 END_IF
        7:
            // disable the external setpoint generator
           physical.processes.disableExtSetGen.start();
           doHoming.state := 8;
        8:
             // wait for the external setpoint generator to be disabled
             IF physical.processes.disableExtSetGen.isIdle() THEN
                 IF physical.processes.disableExtSetGen.isGood() THEN
                    doHoming.state := 9;
                 ELSE
                    doHoming.setActualStatus('Could not disable the external setpoint generator');
                    doHoming.state := 999;
				 END_IF
			 END_IF
        9:
            doHoming.setActualStatus('Enabling LIDA 1 C reset');
            pLida1^.processes.enableCounterResetC.start();
            doHoming.state := 10;
        10:
            IF pLida1^.processes.enableCounterResetC.isIdle() THEN
                IF pLida1^.processes.disableCounterResetC.isGood() THEN
                    doHoming.state := 11;
                ELSE
                    doHoming.setActualStatus('Could not enable LIDA 1 C reset');
                    doHoming.state := 999;
				END_IF
			END_IF
        11:
            doHoming.setActualStatus('Moving until LIDA 1 zero is found');
            pLida1^.updateEnableLatchC(TRUE); // now we can start monitoring the latchCValid flag
            physical.processes.moveRelative.start(distance := homingRange, maxVelocity := homingVelocity);
            doHoming.state := 12;
        12:
            IF pLida1^.latchCValid THEN
                // OK, the counter has been reset!
                physical.processes.stop.start();
                doHoming.state := 13;
            ELSIF physical.processes.moveRelative.isIdle() THEN
                // the end of the range was reached, but the latchCValid was not raised :(
                doHoming.setActualStatus('Could not find the zero mark');
                doHoming.state := 999;
			END_IF
        13:
             // wait for the stop to be finished
             IF virtual.processes.stop.isIdle() THEN
                 IF virtual.processes.stop.isGood() THEN
                    doHoming.state := 14;
                 ELSE
                    doHoming.setActualStatus('Could not stop while traversing the homing range');
                    doHoming.state := 999;
				 END_IF
			 END_IF
        14:
            // disable C latch and C reset 
            doHoming.setActualStatus('Disabling LIDA 1 C reset');
            pLida1^.updateEnableLatchC(FALSE);
            pLida1^.processes.disableCounterResetC.start();
            doHoming.state := 15;
        15:
            IF pLida1^.processes.disableCounterResetC.isIdle() THEN
                IF pLida1^.processes.disableCounterResetC.isGood() THEN
                    doHoming.state := 16;
                ELSE
                    doHoming.setActualStatus('Could not disable LIDA 1 C reset');
                    doHoming.state := 999;
				END_IF
			END_IF
        16:
            doHoming.setActualStatus('Moving back to the zero position');
            physical.processes.moveRelative.start(
                distance := -lida1Position,
                maxVelocity := homingGotoStartVelocity);
            doHoming.state := 17;
        17:
             // wait for the motion to be finished
             IF physical.processes.moveRelative.isIdle() THEN
                 IF physical.processes.moveRelative.isGood() THEN
                    doHoming.state := 18;
                 ELSE
                    doHoming.setActualStatus('Could not move back to the home position');
                    doHoming.state := 999;
				 END_IF
			 END_IF
        18:
            // lida1Position will be now (close to, but not exactly) 0
            // But, it must not be (close to) 0, it must be (close to) the homingHomePosition!
            lida1PositionAfterZeroing := AxesLidaValueToPosition(id := id, encoderValue := pLida1^.counterValue, invert := lidasInvert);
            truePositionAfterZeroing := homingHomePosition + lida1PositionAfterZeroing;
            trueValueAfterZeroing := AxesLidaPositionToValue(id := id, position := truePositionAfterZeroing, invert := lidasInvert);
            
            doHoming.setActualStatus('Synchronizing LIDAs');
            // set the counter FALSE --100ms--> TRUE --100ms--> FALSE
            pLida1^.updateSetCounterValue(trueValueAfterZeroing);
            pLida1^.updateSetCounter(FALSE);
            IF hasLida2() THEN
                pLida2^.updateSetCounterValue(trueValueAfterZeroing);
                pLida2^.updateSetCounter(FALSE);
			END_IF
            IF hasLida3() THEN
                pLida3^.updateSetCounterValue(trueValueAfterZeroing);
                pLida3^.updateSetCounter(FALSE);
			END_IF
            IF hasLida4() THEN
                pLida4^.updateSetCounterValue(trueValueAfterZeroing);
                pLida4^.updateSetCounter(FALSE);
			END_IF
            
            homeTon(IN := FALSE);
            homeTon(IN := TRUE, PT := T#100MS);
            doHoming.state := 19;
        19:
            homeTon(IN := TRUE);
            IF homeTon.Q THEN
                pLida1^.updateSetCounter(TRUE);
                IF hasLida2() THEN
                    pLida2^.updateSetCounter(TRUE);
                END_IF
                IF hasLida3() THEN
                    pLida3^.updateSetCounter(TRUE);
                END_IF
                IF hasLida4() THEN
                    pLida4^.updateSetCounter(TRUE);
                END_IF
                homeTon(IN := FALSE);
                homeTon(IN := TRUE, PT := T#100MS);
                doHoming.state := 20;
			END_IF
        20:
            homeTon(IN := TRUE);
            IF homeTon.Q THEN
                pLida1^.updateSetCounter(FALSE);
                IF hasLida2() THEN
                    pLida2^.updateSetCounter(FALSE);
                END_IF
                IF hasLida3() THEN
                    pLida3^.updateSetCounter(FALSE);
                END_IF
                IF hasLida4() THEN
                    pLida4^.updateSetCounter(FALSE);
                END_IF
                doHoming.state := 21;
			END_IF
        21:
             // synchronize everything with the LIDAs
             setPosition.start(value := lidaAveragePosition);
             doHoming.state := 22;
        22:
             // wait for the new positions to be set
             IF setPosition.isIdle() THEN
                 IF setPosition.isGood() THEN
                    doHoming.state := 23;
                 ELSE
                    doHoming.setActualStatus('Could not update the axis position');
                    doHoming.state := 999;
                 END_IF
             END_IF
        23:     
            // enable the external setpoint generator
            physical.processes.enableExtSetGen.start();
            doHoming.state := 24;
        24:
             // wait for the external setpoint generator to be enabled 
             IF physical.processes.enableExtSetGen.isIdle() THEN
                 IF physical.processes.enableExtSetGen.isGood() THEN
                    doHoming.state := 25;
                 ELSE
                    doHoming.setActualStatus('Could not enable the external setpoint generator');
                    doHoming.state := 999;
				 END_IF
			 END_IF
        25:
            // set the homing flag to TRUE
            physical.processes.forceCalibration.start();
            doHoming.state := 26;
        26:
             // wait for the homing flag to be forced to TRUE
             IF physical.processes.forceCalibration.isIdle() THEN
                 IF physical.processes.forceCalibration.isGood() THEN
                    doHoming.state := 27;
                 ELSE
                    doHoming.setActualStatus('Could not force the calibration flag');
                    doHoming.state := 999;
				 END_IF
			 END_IF
        27:
            // done!
            doHoming.setActualStatus('Homing finished successfully');
            doHoming.state := 1000;
        999:
            // error!
            doHoming.setBad();
            doHoming.setFinished();
            // stop all axes!
            stop.start();
        1000:
            // all done!
            doHoming.setGood();
            doHoming.setFinished();
		
    END_CASE
    
END_IF

METHOD hasLida3 : BOOL
VAR_INPUT
END_VAR
hasLida3 := pLida3 <> 0;
END_METHOD

METHOD hasLida4 : BOOL
VAR_INPUT
END_VAR
hasLida4 := pLida4 <> 0;
END_METHOD

METHOD hasLida2 : BOOL
VAR_INPUT
END_VAR
hasLida2 := pLida2 <> 0;
END_METHOD

METHOD hasLida1 : BOOL
VAR_INPUT
END_VAR
hasLida1 := pLida1 <> 0;
END_METHOD

END_FUNCTION_BLOCK

// ---- MTCS/Common/StateMachines/IncrementalEncoder.TcPOU
FUNCTION_BLOCK IncrementalEncoder EXTENDS SM_IncrementalEncoder
VAR_INPUT
END_VAR
VAR_OUTPUT
END_VAR
VAR
    _adsAddr AT %I* : AMSADDR;
    _adsNetIdStr : STRING;
    _sdoWrite : FB_EcCoeSdoWrite;
    _sdoWriteValue : BOOL;
END_VAR

SUPER^();

THIS^.latchCValid           := status.0;
THIS^.latchExternValid      := status.1;
THIS^.setCounterDone        := status.2;
THIS^.counterUnderflow      := status.3;
THIS^.counterOverflow       := status.4;
THIS^.statusOfInputStatus   := status.5;
THIS^.openCircuit           := status.6;
THIS^.extrapolationStall    := status.7;
THIS^.statusOfInputA        := status.8;
THIS^.statusOfInputB        := status.9;
THIS^.statusOfInputC        := status.10;
THIS^.statusOfInputGate     := status.11;
THIS^.statusOfExternLatch   := status.12;
THIS^.syncError             := status.13;


_adsNetIdStr := CONCAT( BYTE_TO_STRING(_adsAddr.netId[0]),
                 CONCAT( '.',
                  CONCAT( BYTE_TO_STRING(_adsAddr.netId[1]), 
                   CONCAT( '.',
                    CONCAT( BYTE_TO_STRING(_adsAddr.netId[2]), 
                     CONCAT( '.',
                      CONCAT( BYTE_TO_STRING(_adsAddr.netId[3]), 
                       CONCAT( '.',
                        CONCAT( BYTE_TO_STRING(_adsAddr.netId[4]), 
                         CONCAT( '.',
                                 BYTE_TO_STRING(_adsAddr.netId[5])))))))))));

_enableCounterResetC();
_disableCounterResetC();

SUPER^();

METHOD updateSetCounter
VAR_INPUT
    newState : BOOL;
END_VAR
setCounter := newState;
END_METHOD

METHOD _enableCounterResetC
VAR_INPUT
    
END_VAR

IF processes.enableCounterResetC.isBusy() THEN
    
    IF NOT processes.enableCounterResetC.isStarted() THEN
        processes.enableCounterResetC._state := 0;
        processes.enableCounterResetC.setStarted();
	END_IF
    
    CASE processes.enableCounterResetC._state OF
        0:  
            _sdoWriteValue := TRUE;
            _sdoWrite(sNetId     := _adsNetIdStr,
                      nSlaveAddr := _adsAddr.port,
                      bExecute   := FALSE);
            _sdoWrite(sNetId     := _adsNetIdStr,
                      nSlaveAddr := _adsAddr.port,
                      nIndex     := 16#8000,
                      nSubIndex  := 2,
                      pSrcBuf    := ADR(_sdoWriteValue),
                      cbBufLen   := SIZEOF(_sdoWriteValue),
                      bExecute   := TRUE,
                      tTimeout   := DEFAULT_ADS_TIMEOUT);
            processes.enableCounterResetC._state := 1;
        1:
            _sdoWrite(sNetId     := _adsNetIdStr,
                      nSlaveAddr := _adsAddr.port,
                      bExecute   := TRUE);
            IF _sdoWrite.bError THEN
                processes.enableCounterResetC._state := 999;
                processes.enableCounterResetC.setActualStatus(CONCAT('Write error ', UDINT_TO_STRING(_sdoWrite.nErrId)));
            ELSIF NOT _sdoWrite.bBusy THEN
                processes.enableCounterResetC._state := 1000;
			END_IF
            
        999:
            // error!
            processes.enableCounterResetC.setBad();
            processes.enableCounterResetC.setFinished();
        1000:
            // all done!
            processes.enableCounterResetC.setActualStatus('Reset enabled');
            processes.enableCounterResetC.setGood();
            processes.enableCounterResetC.setFinished();
    
	END_CASE
        

END_IF
END_METHOD

METHOD _disableCounterResetC
VAR_INPUT
    
END_VAR

IF processes.disableCounterResetC.isBusy() THEN
    
    IF NOT processes.disableCounterResetC.isStarted() THEN
        processes.disableCounterResetC._state := 0;
        processes.disableCounterResetC.setStarted();
	END_IF
    
    CASE processes.disableCounterResetC._state OF
        0:  
            _sdoWriteValue := FALSE;
            _sdoWrite(sNetId     := _adsNetIdStr,
                      nSlaveAddr := _adsAddr.port,
                      bExecute   := FALSE);
            _sdoWrite(sNetId     := _adsNetIdStr,
                      nSlaveAddr := _adsAddr.port,
                      nIndex     := 16#8000,
                      nSubIndex  := 2,
                      pSrcBuf    := ADR(_sdoWriteValue),
                      cbBufLen   := SIZEOF(_sdoWriteValue),
                      bExecute   := TRUE,
                      tTimeout   := DEFAULT_ADS_TIMEOUT);
            processes.disableCounterResetC._state := 1;
        1:
            _sdoWrite(sNetId     := _adsNetIdStr,
                      nSlaveAddr := _adsAddr.port,
                      bExecute   := TRUE);
            IF _sdoWrite.bError THEN
                processes.disableCounterResetC._state := 999;
                processes.disableCounterResetC.setActualStatus(CONCAT('Write error ', UDINT_TO_STRING(_sdoWrite.nErrId)));
            ELSIF NOT _sdoWrite.bBusy THEN
                processes.disableCounterResetC._state := 1000;
			END_IF
            
        999:
            // error!
            processes.disableCounterResetC.setBad();
            processes.disableCounterResetC.setFinished();
        1000:
            // all done!
            processes.disableCounterResetC.setActualStatus('Reset disabled');
            processes.disableCounterResetC.setGood();
            processes.disableCounterResetC.setFinished();
    
	END_CASE
        

END_IF
END_METHOD

METHOD updateEnableLatchC
VAR_INPUT
    value : BOOL;
END_VAR
enableLatchC := value;
END_METHOD

METHOD updateSetCounterValue
VAR_INPUT
    value : UDINT;
END_VAR
setCounterValue := value;
END_METHOD

END_FUNCTION_BLOCK

// ---- MTCS/Axes/Helper/AxesPowerOnHelper.TcPOU
FUNCTION_BLOCK AxesPowerOnHelper
VAR_INPUT
    id : AxesIds;
    pAblAxis : POINTER TO AngularAxis := 0; (* NULL if no anti-backlash axis is available !!!*)
    pAblDriveChannel : POINTER TO AX52XXDriveChannel := 0; (* NULL if no anti-backlash axis is available !!!*)
    pAblSetpointGenerator : POINTER TO AxesTorqueSetpointGenerator := 0; (* NULL if no anti-backlash axis is available !!!*)
END_VAR
VAR_OUTPUT
END_VAR
VAR_IN_OUT
    setpointGenerator : AxesExternalSetpointGenerator;
    powerOn : AxesPowerOnProcess;
    reset : Process;
    stop     : AxesStopProcess;
    virtual : AngularAxis;
    physical : AngularAxis;
    targetStart : AngularPosition;
END_VAR
VAR
END_VAR

IF powerOn.isBusy() THEN
    
    IF NOT powerOn.isStarted() THEN
        powerOn.state := 0;
        powerOn.setStarted();
	END_IF
    
    CASE powerOn.state OF
        0:
            powerOn.setActualStatus('Starting from unpowered status');
            // first make sure the axes are powered off
            virtual.processes.power.start(enable := FALSE);
            physical.processes.power.start(enable := FALSE);        
            powerOn.state := 1;
        1:
            IF      virtual.processes.power.isIdle() 
                AND physical.processes.power.isIdle() THEN
                
                IF      virtual.processes.power.isGood() 
                   AND  physical.processes.power.isGood() THEN
                    // ok, all axes are disabled
                    powerOn.state := 2;
                ELSE
                    powerOn.setActualStatus('Could not power off the axes!');
                    powerOn.state := 999;
                END_IF
            END_IF
        2:
            powerOn.setActualStatus('Resetting');
            // now we reset the axis first
            reset.start();
            powerOn.state := 3;
        3:
            IF reset.isIdle() THEN
                IF reset.isGood() THEN
                    powerOn.state := 4;
                ELSE
                    powerOn.setActualStatus('Could not reset the axis!');
                    powerOn.state := 999;
				END_IF
			END_IF
        4:
            // now synchronize the virtual axes with the physical axes 
            virtual.processes.setPosition.start(value := physical.axis_ref.NcToPlc.ActPos);
            
            // also synchronize the setpoint generator with the physical axes
            setpointGenerator.synchronize();
            
            powerOn.state := 5;
        5:
            IF  virtual.processes.setPosition.isIdle() THEN
                IF virtual.processes.setPosition.isGood() THEN
                    powerOn.state := 6;
                ELSE
                    powerOn.setActualStatus('Could not synchronize the virtual and physical axes');
                    powerOn.state := 999;
				END_IF
            END_IF
        6:
            powerOn.setActualStatus('Powering on');
            // now power on the axes
            virtual.processes.power.start(enable := TRUE);
            physical.processes.power.start(enable := TRUE);
            powerOn.state := 7;
        7:
            IF      virtual.processes.power.isIdle() 
                AND physical.processes.power.isIdle() THEN
                
                IF      virtual.processes.power.isGood() 
                   AND  physical.processes.power.isGood() THEN
                    // ok, all axes are powered on
                    powerOn.state := 8;
                ELSE
                    powerOn.setActualStatus('Could not power on the axes!');
                    powerOn.state := 999;
                END_IF
            END_IF
        8:
            // now we enable the external setpoint generator
            powerOn.setActualStatus('Enabling external setpoint generator');
            physical.processes.enableExtSetGen.start();
            powerOn.state := 9;
        9:
            // wait for the external setpoint generator to be enabled
            IF physical.processes.enableExtSetGen.isIdle() (* AND ... *) THEN
                IF physical.processes.enableExtSetGen.isGood() THEN
                    powerOn.state := 10;
                ELSE
                    powerOn.state := 999;
                    powerOn.setActualStatus('Could not enable the external setpoint generator');
                END_IF
            END_IF
        10:
            // synchronize the targetStart position
            targetStart(newDegreesValue := physical.axis_ref.PlcToNc.ExtSetPos);
            // now we can turn on the Anti-backlash axis if needed!
            IF hasAblAxis() THEN
                pAblSetpointGenerator^.start();
                pAblAxis^.processes.power.start(enable := TRUE);
                powerOn.state := 11;
            ELSE
                // skip the next step
                powerOn.state := 12;
			END_IF
        11:
            IF pAblAxis^.processes.power.isIdle() THEN
                IF  pAblAxis^.processes.power.isGood() THEN
                    // ok, all axes are powered on
                    powerOn.state := 12;
                ELSE
                    powerOn.setActualStatus('Could not power on the anti-backlash axis!');
                    powerOn.state := 999;
                END_IF
            END_IF
        12:
            // all done!
            powerOn.state := 1000;
        999:
            // error!
            powerOn.setBad();
            powerOn.setFinished();
            // stop all axes
            stop.start();
            IF hasAblAxis() THEN
                // remove the ABL torque
                pAblSetpointGenerator^.stop();
			END_IF
        1000:
            // ok done
            powerOn.setFinished();
            powerOn.setGood();
            powerOn.setActualStatus('Powered on');
    END_CASE
    
END_IF

METHOD hasAblAxis : BOOL
VAR_INPUT
END_VAR
hasAblAxis := (pAblAxis <> 0) AND (pAblDriveChannel <> 0) AND (pAblSetpointGenerator <> 0);
END_METHOD

END_FUNCTION_BLOCK

// ---- MTCS/Common/StateMachines/AngularPosition.TcPOU
FUNCTION_BLOCK AngularPosition EXTENDS SM_AngularPosition
VAR_INPUT
END_VAR
VAR_OUTPUT
END_VAR
VAR
    _testVar : INT;
END_VAR

SUPER^();



// do stuff

//SUPER^();

END_FUNCTION_BLOCK

// ---- MTCS/Axes/Helper/AxesStopHelper.TcPOU
FUNCTION_BLOCK AxesStopHelper
VAR_INPUT
END_VAR
VAR_OUTPUT
END_VAR
VAR_IN_OUT
    setpointGenerator : AxesExternalSetpointGenerator;
    stop     : AxesStopProcess;
    virtual : AngularAxis;
    physical : AngularAxis;
END_VAR
VAR
END_VAR

IF stop.isBusy() THEN
    
    IF NOT stop.isStarted() THEN
        stop.state := 0;
        stop.setStarted();
	END_IF
    
    // two cases are possible:
    //  1) the external setpoint generator is enabled
    //     --> 1.a) synchronize the virtual with the physical axis
    //         1.b) stop tracking
    //         1.c) stop the virtual axis (even if it was not moving)
    //  2) the external setpoint generator is disabled
    //     --> 2.a) stop both the physical axis and the virtual axis (even if they were not moving)'
    //  
    //  Either case, if they fail to stop, we power off the axes
    
    CASE stop.state OF
        0:
            stop.setActualStatus('Now stopping'); 
            IF physical.axis_ref.Status.ExtSetPointGenEnabled THEN
                // case 1.a) synchronize the virtual with the physical axis
                virtual.processes.setPosition.start(value := physical.axis_ref.NcToPlc.ActPos);
                stop.state := 1;
            ELSE
                // case 2.a) stop both the physical axis and the virtual axis (even if they were not moving)
                physical.processes.stop.start();
                virtual.processes.stop.start(); // not needed in fact, but it's better to make sure it is stopped too
                stop.state := 3;
			END_IF
        1:
            IF virtual.processes.setPosition.isIdle() THEN
                // regardless of whether the stopping worked or not go to the next step
                // 1.b) stop tracking
                setpointGenerator.stopTracking();
                // 1.c) stop the virtual axis (even if it was not moving)
                virtual.processes.stop.start();
                stop.state := 2;
			END_IF
        2:
            IF virtual.processes.stop.isIdle() THEN
                IF virtual.processes.stop.isGood() THEN
                    stop.state := 1000;
                ELSE
                    stop.setActualStatus('Could not stop the virtual axis');
                    stop.state := 999;
                END_IF
            END_IF
        3:
            IF      physical.processes.stop.isIdle()
                AND virtual.processes.stop.isIdle() 
            THEN
                IF     physical.processes.stop.isGood()
                   AND virtual.processes.stop.isGood() 
                THEN
                    stop.state := 1000;
                ELSE
                    stop.setActualStatus('Could not stop the physical and virtual axes');
                    stop.state := 999;
                END_IF
			END_IF
        1000:
            // ok done
            stop.setFinished();
            stop.setGood();
            stop.setActualStatus('Stopped');
        999:
            // error!
            // try to power off the motors
            stop.setBad();
            stop.state := 9991;
        9991:
            physical.processes.power.start(enable := FALSE);
            virtual.processes.power.start(enable := FALSE);
        9992:
            // still in error, nothing to do
            stop.setFinished();
            
    END_CASE
    
END_IF

END_FUNCTION_BLOCK

// ---- MTCS/Axes/Helper/AxesSetPositionHelper.TcPOU
FUNCTION_BLOCK AxesSetPositionHelper
VAR_INPUT
END_VAR
VAR_OUTPUT
END_VAR
VAR_IN_OUT
    setpointGenerator : AxesExternalSetpointGenerator;
    setPosition :  AxesSetpositionProcess;;
    virtual : AngularAxis;
    physical : AngularAxis;
END_VAR
VAR
    _ton : TON;
END_VAR

IF setPosition.isBusy() THEN
    
    IF NOT setPosition.isStarted() THEN
        setPosition._state := 0;
        setPosition.setStarted();
	END_IF
    
    CASE setPosition._state OF
        0:
            setPosition.setActualStatus('Setting the position'); 
            IF physical.axis_ref.Status.ExtSetPointGenEnabled THEN
                setPosition.setActualStatus('Cannot set position if ExtSetGen is enabled!');
                setPosition._state := 999;
            ELSE
                setPosition._state := 1;
			END_IF
        1:
             // set the positions
             virtual.processes.setPosition.start(value := setPosition.get.value);
             physical.processes.setPosition.start(value := setPosition.get.value);
             setpointGenerator.setPosition(setPosition.get.value);
             // WARNING: even if setPosition becomes idle, then the ActPos of the axis is not adjusted yet for 2 cycles!
             // So it takes some more cycles after setPosition, for the ActPos to become the new value
             // Therefore, we wait a small time 
             _ton(IN := FALSE);
             _ton(IN := TRUE, PT := T#50MS);
             setPosition._state := 2;
        2:
             _ton(IN := TRUE);
             IF _ton.Q THEN
                 // wait for the new positions to be set
                 IF physical.processes.setPosition.isIdle() AND virtual.processes.setPosition.isIdle() THEN
                     IF physical.processes.setPosition.isGood() AND virtual.processes.setPosition.isGood() THEN
                        setPosition._state := 1000;
                     ELSE
                        setPosition.setActualStatus('Could not set physical and virtual position');
                        setPosition._state := 999;
                     END_IF
                 END_IF
			 END_IF
        999:
            // error!
            // try to power off the motors
            setPosition.setBad();
            setPosition.setFinished();
        1000:
            // ok done
            setPosition.setFinished();
            setPosition.setGood();
            setPosition.setActualStatus('Position was set');

            
    END_CASE
    
END_IF

END_FUNCTION_BLOCK

// ---- MTCS/Axes/Helper/AxesCalculateTorqueCommandValue.TcPOU
FUNCTION AxesCalculateTorqueCommandValue : INT
VAR_INPUT
    torqueSetpoint : LREAL; // Nm
    torqueConstant : LREAL; // Nm/A
    channelPeakCurrent : LREAL; // A
END_VAR
VAR
    currentAtMotor : LREAL; // A
    currentFraction : LREAL; // [0.0..1.0]
END_VAR


IF torqueConstant <> 0 THEN
    currentAtMotor := torqueSetpoint / torqueConstant;
ELSE
    currentAtMotor := 0.0;
END_IF

IF channelPeakCurrent <> 0 THEN
    currentFraction := currentAtMotor / channelPeakCurrent;
ELSE
    currentFraction := 0.0;
END_IF

AxesCalculateTorqueCommandValue := LREAL_TO_INT(currentFraction * 1000.0); // units: tenth of a percent ]]>

END_FUNCTION

// ---- MTCS/Axes/Helper/RAD_TO_HOUR.TcPOU
FUNCTION RAD_TO_HOUR : LREAL
VAR_INPUT
    rad : LREAL;
END_VAR
VAR
END_VAR

RAD_TO_HOUR := rad * 12.0 / PI;

END_FUNCTION

// ---- MTCS/Axes/StateMachines/AxesElevationAxis.TcPOU
FUNCTION_BLOCK AxesElevationAxis EXTENDS SM_AxesElevationAxis
VAR_INPUT
END_VAR
VAR_OUTPUT
END_VAR
VAR
    // setpoint generator
	{attribute 'OPC.UA.DA' := '0'}
    _setGen : AxesExternalSetpointGenerator;
    
    // helpers
	{attribute 'OPC.UA.DA' := '0'}
    _powerOnHelper : AxesPowerOnHelper;
	{attribute 'OPC.UA.DA' := '0'}
    _powerOffHelper : AxesPowerOffHelper;
	{attribute 'OPC.UA.DA' := '0'}
    _homingHelper : AxesHomingHelper;
	{attribute 'OPC.UA.DA' := '0'}
    _moveOutOfLimitSwitchHelper : AxesMoveOutOfLimitSwitchHelper;
	{attribute 'OPC.UA.DA' := '0'}
    _stopHelper : AxesStopHelper;
	{attribute 'OPC.UA.DA' := '0'}
    _quickStopHelper : AxesQuickStopHelper;
	{attribute 'OPC.UA.DA' := '0'}
    _setPositionHelper : AxesSetPositionHelper;
	{attribute 'OPC.UA.DA' := '0'}
    _unlockBrakeHelper : AxesUnlockBrakeHelper;
    
    // RMS and average setpoint deviation calculator
	{attribute 'OPC.UA.DA' := '0'}
    _deviationCalculator: AverageAndRmsCalculator;
    // local copy of the isTracking flag
	{attribute 'OPC.UA.DA' := '0'}
    _isTracking: BOOL;
END_VAR

_update();

_resetting();

_powerOnHelper(
    id                      := id,
    setpointGenerator       := _setGen,
    powerOn                 := processes.powerOn,
    stop                    := processes.stop,
    reset                   := processes.reset,
    virtual                 := parts.virtualAxis,
    physical                := parts.physicalAxis,
    targetStart             := targetStart,
    pAblAxis                := 0,
    pAblDriveChannel        := 0,
    pAblSetpointGenerator   := 0);

_powerOffHelper(
    setpointGenerator       := _setGen,
    powerOff                := processes.powerOff,
    stop                    := processes.stop,
    virtual                 := parts.virtualAxis,
    physical                := parts.physicalAxis,
    pAblAxis                := 0,
    pAblDriveChannel        := 0,
    pAblSetpointGenerator   := 0);

_moveOutOfLimitSwitchHelper(
    setpointGenerator               := _setGen,
    positiveLimitSwitchError        := positiveLimitSwitchError,
    negativeLimitSwitchError        := negativeLimitSwitchError,
    positiveLimitSwitchInput        := config.positiveLimitSwitchInput,
    negativeLimitSwitchInput        := config.negativeLimitSwitchInput,
    moveOutOfLimitSwitchDistance    := config.moveOutOfLimitSwitchDistance,
    moveOutOfLimitSwitch            := processes.moveOutOfLimitSwitch,
    moveRelative                    := processes.moveRelative,
    powerOn                         := processes.powerOn,
    reset                           := processes.reset,
    virtual                         := parts.virtualAxis,
    physical                        := parts.physicalAxis,
    driveChannel                    := mainDriveChannel);


_homingHelper(
    homingStartAbsEncPosition   := config.homingStartAbsEncPosition,
    homingVelocity              := config.homingVelocity,
    homingRange                 := config.homingRange,
    homingGotoStartVelocity     := config.homingGotoStartVelocity,
    homingHomePosition          := config.homingHomePosition,
    lidasInvert                 := config.lidasInvert,
    absoluteEncoderPosition     := absoluteEncoderPosition.degrees.value,
    lidaAveragePosition         := lidaAveragePosition.degrees.value,
    lida1Position               := lida1Position.degrees.value,
    setpointGenerator           := _setGen,
    doHoming                    := processes.doHoming,
    stop                        := processes.stop,
    setPosition                 := processes.setPosition,
    virtual                     := parts.virtualAxis,
    physical                    := parts.physicalAxis,
    pLida1                      := ADR(parts.lida1),
    pLida2                      := ADR(parts.lida2),
    pLida3                      := 0,
    pLida4                      := 0);

_moveAbsolute();
_moveRelative();
_moveVelocity();

_stopHelper(
    setpointGenerator   := _setGen,
    stop                := processes.stop,
    virtual             := parts.virtualAxis,
    physical            := parts.physicalAxis);
    
_quickStopHelper(
    deceleration        := config.quickStopDeceleration, 
    jerk                := config.quickStopJerk,
    setpointGenerator   := _setGen,
    quickStop           := processes.quickStop,
    virtual             := parts.virtualAxis,
    physical            := parts.physicalAxis);

_setPositionHelper(
    setpointGenerator   := _setGen,
    setPosition         := processes.setPosition,
    virtual             := parts.virtualAxis,
    physical            := parts.physicalAxis);

_unlockBrakeHelper(
    unlockBrake         := processes.unlockBrake,
    driveChannel        := driveChannel);

_update();

METHOD _update : LREAL
VAR_INPUT
END_VAR
VAR
    absoluteEncoderReduction : LREAL;
END_VAR
// update the superclass
SUPER^(
    config := config,
    driveChannel := driveChannel,
    mainDriveChannel := mainDriveChannel);

// update the limit switches
positiveLimitSwitchError := NOT GETBIT32(inVal32 := INT_TO_DWORD(driveChannel.digitalInputs), bitNo := config.positiveLimitSwitchInput);
negativeLimitSwitchError := NOT GETBIT32(inVal32 := INT_TO_DWORD(driveChannel.digitalInputs), bitNo := config.negativeLimitSwitchInput);

// update the LIDA positions
lida1Position(newDegreesValue := AxesLidaValueToPosition(id := AxesIds.AZI, encoderValue := parts.lida1.counterValue, invert := config.lidasInvert));
lida2Position(newDegreesValue := AxesLidaValueToPosition(id := AxesIds.AZI, encoderValue := parts.lida2.counterValue, invert := config.lidasInvert));

// calculate the average value
lidaAveragePosition( newDegreesValue := 
    AxesCalculateLidaAveragePosition(
        lida1Position := lida1Position.degrees.value,
        lida2Position := lida2Position.degrees.value,
        lida3Position := 0.0,
        lida4Position := 0.0,
        useLida1      := NOT (parts.lida1.openCircuit OR parts.lida1.syncError OR parts.lida1.extrapolationStall), 
        useLida2      := NOT (parts.lida2.openCircuit OR parts.lida2.syncError OR parts.lida2.extrapolationStall),
        useLida3      := FALSE,
        useLida4      := FALSE));

// update the absolute encoder position
IF  config.absoluteEncoderInvert THEN
    absoluteEncoderReduction := -REDUCTION_ABS_ENC_TO_TEL;
ELSE
    absoluteEncoderReduction := REDUCTION_ABS_ENC_TO_TEL;
END_IF
absoluteEncoderPosition(newDegreesValue := AxesSSIValueToPosition(
        reduction       := absoluteEncoderReduction,
        encoderValue    := parts.absoluteEncoder.counterValue,
        zeroOffset      := config.absoluteEncoderOffset));

// update the actual position/velocity/acceleration
actPos(newDegreesValue := parts.physicalAxis.axis_ref.NcToPlc.ActPos);
actVelo(newDegreesPerSecondValue := parts.physicalAxis.axis_ref.NcToPlc.ActVelo);
actAcc(newDegreesPerSquareSecondValue := parts.physicalAxis.axis_ref.NcToPlc.ActAcc);
setPos(newDegreesValue := parts.physicalAxis.axis_ref.NcToPlc.SetPos);
setVelo(newDegreesPerSecondValue := parts.physicalAxis.axis_ref.NcToPlc.SetVelo);
setAcc(newDegreesPerSquareSecondValue := parts.physicalAxis.axis_ref.NcToPlc.SetAcc);
IF parts.physicalAxis.axis_ref.Status.ExtSetPointGenEnabled THEN
    targetPos(newDegreesValue := parts.physicalAxis.axis_ref.PlcToNc.ExtSetPos);
    targetOffset(newDegreesValue := parts.virtualAxis.actPos.degrees.value - targetStart.degrees.value);
ELSE
    targetPos(newDegreesValue := parts.physicalAxis.axis_ref.NcToPlc.TargetPos);
    targetOffset(newDegreesValue := 0.0);
END_IF

// update the actual torque feedback on the telescope side
actTorque(newNewtonmeterValue := driveChannel.actualTorqueFeedback.newtonmeter.value * 1440);
END_METHOD

METHOD _moveVelocity
VAR_INPUT
END_VAR
VAR
    velocityDegPerSec : LREAL;
END_VAR
IF processes.moveVelocity.isBusy() THEN
    
    IF NOT processes.moveVelocity.isStarted() THEN
        
        velocityDegPerSec := AxesMoveVelocityUnitsToDegPerSec(units := processes.moveVelocity.get.units, value := processes.moveVelocity.get.value);
        
        parts.virtualAxis.processes.moveVelocity.start(value := velocityDegPerSec);
    
        processes.moveVelocity.setStarted();
            
	END_IF

    // update the statuses
    processes.moveVelocity.statuses.busyStatus(isBusy := parts.virtualAxis.processes.moveVelocity.statuses.busyStatus.isBusy);
    processes.moveVelocity.statuses.healthStatus(
        isGood := parts.virtualAxis.processes.moveVelocity.statuses.healthStatus.isGood,
        hasWarning := parts.virtualAxis.processes.moveVelocity.statuses.healthStatus.hasWarning);
    processes.moveVelocity.setActualStatus(parts.virtualAxis.processes.moveVelocity.actualStatus);

END_IF
END_METHOD

METHOD _resetting : LREAL
VAR_INPUT
END_VAR
IF processes.reset.isBusy() THEN
    
    IF NOT processes.reset.isStarted() THEN
        processes.reset._state := 0;
        processes.reset.setStarted();
	END_IF
    
    CASE processes.reset._state OF
        0:
            // reset all processes so that they are green again
            processes.doHoming.resetIfIdle();
            processes.moveAbsolute.resetIfIdle();
            processes.moveOutOfLimitSwitch.resetIfIdle();
            processes.moveRelative.resetIfIdle();
            processes.moveVelocity.resetIfIdle();
            processes.powerOff.resetIfIdle();
            processes.powerOn.resetIfIdle();
            processes.quickStop.resetIfIdle();
            processes.setPosition.resetIfIdle();
            processes.stop.resetIfIdle();
            processes.unlockBrake.resetIfIdle();
            
